// Create log entry for AccelerationRate
CreateLogMessagePara1 ( Timestamp   := AxesGroup.InternalData.SystemTime,
                        MessageType := MessageType.CMD,
                        Severity    := Severity.DEBUG,
                        MessageCode := 0,
                        MessageText := 'Command.AccelerationRate = {1}',
                        Para1       :=  UINT_TO_STRING(_command.AccelerationRate));
                        
// Create log entry for DecelerationRate
CreateLogMessagePara1 ( Timestamp   := AxesGroup.InternalData.SystemTime,
                        MessageType := MessageType.CMD,
                        Severity    := Severity.DEBUG,
                        MessageCode := 0,
                        MessageText := 'Command.DecelerationRate = {1}',
                        Para1       :=  UINT_TO_STRING(_command.DecelerationRate));

// Create log entry for JerkRate
CreateLogMessagePara1 ( Timestamp   := AxesGroup.InternalData.SystemTime,
                        MessageType := MessageType.CMD,
                        Severity    := Severity.DEBUG,
                        MessageCode := 0,
                        MessageText := 'Command.JerkRate = {1}',
                        Para1       :=  UINT_TO_STRING(_command.JerkRate));

// Create log entry for ToolNo
CreateLogMessagePara1 ( Timestamp   := AxesGroup.InternalData.SystemTime,
                        MessageType := MessageType.CMD,
                        Severity    := Severity.DEBUG,
                        MessageCode := 0,
                        MessageText := 'Command.ToolNo = {1}',
                        Para1       :=  USINT_TO_STRING(_command.ToolNo));

// Create log entry for FrameNo
CreateLogMessagePara1 ( Timestamp   := AxesGroup.InternalData.SystemTime,
                        MessageType := MessageType.CMD,
                        Severity    := Severity.DEBUG,
                        MessageCode := 0,
                        MessageText := 'Command.FrameNo = {1}',
                        Para1       :=  USINT_TO_STRING(_command.FrameNo));

// Create log entry for BlendingMode
CreateLogMessagePara1 ( Timestamp   := AxesGroup.InternalData.SystemTime,
                        MessageType := MessageType.CMD,
                        Severity    := Severity.DEBUG,
                        MessageCode := 0,
                        MessageText := 'Command.BlendingMode = {1}',
                        Para1       :=  BLENDING_MODE_TO_STRING(_command.BlendingMode));

// Create log entry for Reserve
CreateLogMessagePara1 ( Timestamp   := AxesGroup.InternalData.SystemTime,
                        MessageType := MessageType.CMD,
                        Severity    := Severity.DEBUG,
                        MessageCode := 0,
                        MessageText := 'Command.Reserve = {1}',
                        Para1       :=  BYTE_TO_STRING(_command.Reserve));

// Create log entry for BlendingParameter[0]
CreateLogMessagePara1 ( Timestamp   := AxesGroup.InternalData.SystemTime,
                        MessageType := MessageType.CMD,
                        Severity    := Severity.DEBUG,
                        MessageCode := 0,
                        MessageText := 'Command.BlendingParameter[0] = {1}',
                        Para1       :=  REAL_TO_STRING(_command.BlendingParameter[0]));

// Create log entry for BlendingParameter[1]
CreateLogMessagePara1 ( Timestamp   := AxesGroup.InternalData.SystemTime,
                        MessageType := MessageType.CMD,
                        Severity    := Severity.DEBUG,
                        MessageCode := 0,
                        MessageText := 'Command.BlendingParameter[1] = {1}',
                        Para1       :=  REAL_TO_STRING(_command.BlendingParameter[1]));

// Create log entry for Position.X
CreateLogMessagePara1 ( Timestamp   := AxesGroup.InternalData.SystemTime,
                        MessageType := MessageType.CMD,
                        Severity    := Severity.DEBUG,
                        MessageCode := 0,
                        MessageText := 'Command.Position.X = {1}',
                        Para1       :=  REAL_TO_STRING(_command.Position.X));

// Create log entry for Position.Y
CreateLogMessagePara1 ( Timestamp   := AxesGroup.InternalData.SystemTime,
                        MessageType := MessageType.CMD,
                        Severity    := Severity.DEBUG,
                        MessageCode := 0,
                        MessageText := 'Command.Position.Y = {1}',
                        Para1       :=  REAL_TO_STRING(_command.Position.Y));

// Create log entry for Position.Z
CreateLogMessagePara1 ( Timestamp   := AxesGroup.InternalData.SystemTime,
                        MessageType := MessageType.CMD,
                        Severity    := Severity.DEBUG,
                        MessageCode := 0,
                        MessageText := 'Command.Position.Z = {1}',
                        Para1       :=  REAL_TO_STRING(_command.Position.Z));

// Create log entry for Position.Rx
CreateLogMessagePara1 ( Timestamp   := AxesGroup.InternalData.SystemTime,
                        MessageType := MessageType.CMD,
                        Severity    := Severity.DEBUG,
                        MessageCode := 0,
                        MessageText := 'Command.Position.Rx = {1}',
                        Para1       :=  REAL_TO_STRING(_command.Position.Rx));

// Create log entry for Position.Ry
CreateLogMessagePara1 ( Timestamp   := AxesGroup.InternalData.SystemTime,
                        MessageType := MessageType.CMD,
                        Severity    := Severity.DEBUG,
                        MessageCode := 0,
                        MessageText := 'Command.Position.Ry = {1}',
                        Para1       :=  REAL_TO_STRING(_command.Position.Ry));

// Create log entry for Position.Rz
CreateLogMessagePara1 ( Timestamp   := AxesGroup.InternalData.SystemTime,
                        MessageType := MessageType.CMD,
                        Severity    := Severity.DEBUG,
                        MessageCode := 0,
                        MessageText := 'Command.Position.Rz = {1}',
                        Para1       :=  REAL_TO_STRING(_command.Position.Rz));

// Create log entry for Position.Config
CreateLogMessagePara1 ( Timestamp   := AxesGroup.InternalData.SystemTime,
                        MessageType := MessageType.CMD,
                        Severity    := Severity.DEBUG,
                        MessageCode := 0,
                        MessageText := 'Command.Config = {1}',
                        Para1       :=  ARM_CONFIG_TO_STRING(_command.Position.Config));

// Create log entry for Position.Reserve
CreateLogMessagePara1 ( Timestamp   := AxesGroup.InternalData.SystemTime,
                        MessageType := MessageType.CMD,
                        Severity    := Severity.DEBUG,
                        MessageCode := 0,
                        MessageText := 'Command.Position.Reserve = {1}',
                        Para1       :=  BYTE_TO_STRING(_command.Reserve));

// Create log entry for Position.TurnNumber[0]
CreateLogMessagePara1 ( Timestamp   := AxesGroup.InternalData.SystemTime,
                        MessageType := MessageType.CMD,
                        Severity    := Severity.DEBUG,
                        MessageCode := 0,
                        MessageText := 'Command.Position.TurnNumber[0] = {1}',
                        Para1       :=  BYTE_TO_STRING(CombineHalfSints(HalfSintHi := _command.Position.TurnNumber.J2Turns, 
                                                                        HalfSintLo := _command.Position.TurnNumber.J1Turns)));

// Create log entry for Position.TurnNumber[1]
CreateLogMessagePara1 ( Timestamp   := AxesGroup.InternalData.SystemTime,
                        MessageType := MessageType.CMD,
                        Severity    := Severity.DEBUG,
                        MessageCode := 0,
                        MessageText := 'Command.Position.TurnNumber[1] = {1}',
                        Para1       :=  BYTE_TO_STRING(CombineHalfSints(HalfSintHi := _command.Position.TurnNumber.J4Turns,
                                                                        HalfSintLo := _command.Position.TurnNumber.J3Turns)));

// Create log entry for Position.TurnNumber[2]
CreateLogMessagePara1 ( Timestamp   := AxesGroup.InternalData.SystemTime,
                        MessageType := MessageType.CMD,
                        Severity    := Severity.DEBUG,
                        MessageCode := 0,
                        MessageText := 'Command.Position.TurnNumber[2] = {1}',
                        Para1       :=  BYTE_TO_STRING(CombineHalfSints(HalfSintHi := _command.Position.TurnNumber.J6Turns,
                                                                        HalfSintLo := _command.Position.TurnNumber.J5Turns)));


// Create log entry for Position.TurnNumber[3]
CreateLogMessagePara1 ( Timestamp   := AxesGroup.InternalData.SystemTime,
                        MessageType := MessageType.CMD,
                        Severity    := Severity.DEBUG,
                        MessageCode := 0,
                        MessageText := 'Command.Position.TurnNumber[3] = {1}',
                        Para1       :=  SINT_TO_STRING(_command.Position.TurnNumber.E1Turns));

// Create log entry for Position.E1
CreateLogMessagePara1 ( Timestamp   := AxesGroup.InternalData.SystemTime,
                        MessageType := MessageType.CMD,
                        Severity    := Severity.DEBUG,
                        MessageCode := 0,
                        MessageText := 'Command.Position.E1 = {1}',
                        Para1       :=  REAL_TO_STRING(_command.Position.E1));

// Create log entry for Manipulation
CreateLogMessagePara1 ( Timestamp   := AxesGroup.InternalData.SystemTime,
                        MessageType := MessageType.CMD,
                        Severity    := Severity.DEBUG,
                        MessageCode := 0,
                        MessageText := 'Command.Manipulation = {1}',
                        Para1       :=  BOOL_TO_STRING(_command.Manipulation));

// Create log entry for TurnMode
CreateLogMessagePara1 ( Timestamp   := AxesGroup.InternalData.SystemTime,
                        MessageType := MessageType.CMD,
                        Severity    := Severity.DEBUG,
                        MessageCode := 0,
                        MessageText := 'Command.TurnMode = {1}',
                        Para1       :=  TURN_MODE_TO_STRING(_command.TurnMode));

// Create log entry for ConfigMode[0]
CreateLogMessagePara1 ( Timestamp   := AxesGroup.InternalData.SystemTime,
                        MessageType := MessageType.CMD,
                        Severity    := Severity.DEBUG,
                        MessageCode := 0,
                        MessageText := 'Command.ConfigMode[0] = {1}',
                        Para1       :=  BYTE_TO_STRING_BIN(_command.ConfigMode[0]));

// Create log entry for ConfigMode[1]
CreateLogMessagePara1 ( Timestamp   := AxesGroup.InternalData.SystemTime,
                        MessageType := MessageType.CMD,
                        Severity    := Severity.DEBUG,
                        MessageCode := 0,
                        MessageText := 'Command.ConfigMode[1] = {1}',
                        Para1       :=  BYTE_TO_STRING_BIN(_command.ConfigMode[1]));

// Create log entry for Reserve3
CreateLogMessagePara1 ( Timestamp   := AxesGroup.InternalData.SystemTime,
                        MessageType := MessageType.CMD,
                        Severity    := Severity.DEBUG,
                        MessageCode := 0,
                        MessageText := 'Command.Reserve3 = {1}',
                        Para1       :=  BYTE_TO_STRING(_command.Reserve3));

// Create log entry for Reserve4
CreateLogMessagePara1 ( Timestamp   := AxesGroup.InternalData.SystemTime,
                        MessageType := MessageType.CMD,
                        Severity    := Severity.DEBUG,
                        MessageCode := 0,
                        MessageText := 'Command.Reserve4 = {1}',
                        Para1       :=  BYTE_TO_STRING(_command.Reserve4));

// Create log entry for MoveTime
CreateLogMessagePara1 ( Timestamp   := AxesGroup.InternalData.SystemTime,
                        MessageType := MessageType.CMD,
                        Severity    := Severity.DEBUG,
                        MessageCode := 0,
                        MessageText := 'Command.MoveTime = {1}',
                        Para1       :=  UINT_TO_STRING(_command.MoveTime));

// Create log entry for Position.E2
CreateLogMessagePara1 ( Timestamp   := AxesGroup.InternalData.SystemTime,
                        MessageType := MessageType.CMD,
                        Severity    := Severity.DEBUG,
                        MessageCode := 0,
                        MessageText := 'Command.Position.E2 = {1}',
                        Para1       :=  REAL_TO_STRING(_command.Position.E2));

// Create log entry for Position.E3
CreateLogMessagePara1 ( Timestamp   := AxesGroup.InternalData.SystemTime,
                        MessageType := MessageType.CMD,
                        Severity    := Severity.DEBUG,
                        MessageCode := 0,
                        MessageText := 'Command.Position.E3 = {1}',
                        Para1       :=  REAL_TO_STRING(_command.Position.E3));

// Create log entry for Position.E4
CreateLogMessagePara1 ( Timestamp   := AxesGroup.InternalData.SystemTime,
                        MessageType := MessageType.CMD,
                        Severity    := Severity.DEBUG,
                        MessageCode := 0,
                        MessageText := 'Command.Position.E4 = {1}',
                        Para1       :=  REAL_TO_STRING(_command.Position.E4));

// Create log entry for Position.E5
CreateLogMessagePara1 ( Timestamp   := AxesGroup.InternalData.SystemTime,
                        MessageType := MessageType.CMD,
                        Severity    := Severity.DEBUG,
                        MessageCode := 0,
                        MessageText := 'Command.Position.E5 = {1}',
                        Para1       :=  REAL_TO_STRING(_command.Position.E5));

// Create log entry for Position.E6
CreateLogMessagePara1 ( Timestamp   := AxesGroup.InternalData.SystemTime,
                        MessageType := MessageType.CMD,
                        Severity    := Severity.DEBUG,
                        MessageCode := 0,
                        MessageText := 'Command.Position.E6 = {1}',
                        Para1       :=  REAL_TO_STRING(_command.Position.E6));
END_METHOD

METHOD FB_init : BOOL
VAR_INPUT
  /// if TRUE, the retain variables are initialized (warm start / cold start)
  bInitRetains : BOOL; 
  /// if TRUE, the instance afterwards gets moved into the copy code (online change)
  bInCopyCode  : BOOL;  
END_VAR
MyType := 'MC_MoveDirectAbsoluteFB';
END_METHOD

METHOD PROTECTED OnCall
VAR_IN_OUT
  /// Robot assignment of function
  AxesGroup : AxesGroup; 
END_VAR
// call base implementation
SUPER^.OnCall(AxesGroup := AxesGroup);

CASE _stepCmd OF
  
  00:  IF ( _execute_R.Q )  
       THEN
         // Check function is supported and parameter are valid ?
         IF (( CheckFunctionSupported( AxesGroup := AxesGroup )) AND
             ( CheckParameterValid   ( AxesGroup := AxesGroup )))      
         THEN
           // set busy flag
           Busy := TRUE;
           // Reset command outputs
           SysDepMemSet(pDest := ADR(OutCmd), Value := 0, DataLen := SIZEOF(OutCmd));         
           // apply command parameter
          _parCmd := ParCmd;
           // init parameter sequence
          _command.ParSeq := 1;
           // create command data
           CommandData := CreateCommandPayload(AxesGroup := AxesGroup);
           // Add command to active command register
          _uniqueID := AxesGroup.Acyclic.ActiveCommandRegister.AddCmd( pCommandFB := ADR(THIS^ ));     
           // set timeout
           SetTimeout(PT := _timeoutCmd, rTimer := _timerCmd);
           // inc step counter
          _stepCmd := _stepCmd + 1;
         END_IF 
       END_IF
     

  01:  // Wait for responce received
       IF ( _responseReceived )
       THEN
         // reset response received flag
        _responseReceived := FALSE;
         // reset Active flag
         Active := FALSE;
         
         CASE  _response.State 
         OF
           CmdMessageState.BUFFERED    : CommandBuffered    := TRUE;
           CmdMessageState.ACTIVE      : Active             := TRUE;
           CmdMessageState.INTERRUPTED : CommandInterrupted := TRUE;           
           CmdMessageState.DONE        : Done               := TRUE;           
           CmdMessageState.ABORTED     : CommandAborted     := TRUE;
           CmdMessageState.ERROR       : Error              := TRUE;
         END_CASE
                
         // Done, Aborted or Error ?
         IF (_response.State >= CmdMessageState.DONE )
         THEN
           // Reset Busy flag
           Busy := FALSE;
           // Update results
           OutCmd.Progress          := _response.Progress;
           OutCmd.FollowID          := _response.OriginID;
           OutCmd.RemainingDistance := _response.RemainingDistance;
           // set timeout
           SetTimeout(PT := _timeoutCmd, rTimer := _timerCmd);
           // inc step counter
          _stepCmd := _stepCmd + 1; 
         END_IF
       END_IF


  02: IF ( NOT Execute)
      THEN
        Reset();
      END_IF     

ELSE
  // invalid step
  ErrorID := RobotLibraryEvents.ERR_INVALID_STEP;
END_CASE


// Reset FB
IF ( NOT Execute )
THEN
  Reset();
END_IF
END_METHOD

METHOD INTERNAL ParseResponsePayload : DINT
VAR_INPUT
  /// Response data
  ResponseData : RobotLibraryRecvDataFB;
  /// Timestamp
  Timestamp    : SystemTime;  
END_VAR
// Table 6-255: Received CMD payload (RC to PLC) of "MoveDirectAbsolute"
// --------------------------
// Header
// --------------------------
// Byte 00 : USINT   - ParSeq | State     
// Byte 01 : SINT    - AlarmMessageSeverity    
// Byte 02 : UINT    - AlarmMessageCode HB
// Byte 03 :         - AlarmMessageCode LB
// --------------------------
// Datablock
// --------------------------
// Byte 04 : USINT      - InvocationCounter
// Byte 05 : SINT       - Reserved
// Byte 06 : INT        - OriginID HW HB
// Byte 07 :            - OriginID HW LB
// Byte 08 : UINT       - Progress HW HB
// Byte 09 :            - Progress HW LB
// Byte 10 : REAL       - RemainingDistance HW HB
// Byte 11 :            - RemainingDistance HW LB
// Byte 12 :            - RemainingDistance LW HB
// Byte 13 :            - RemainingDistance LW LB
// call base implementation to parse the header from payload buffer
ResponseData.PayloadPtr := SUPER^.ParseResponsePayload(ResponseData := ResponseData, Timestamp := Timestamp);

// copy parsed header to response
_response.ParSeq               := _rspHeader.ParSeq;
_response.State                := _rspHeader.State;
_response.AlarmMessageSeverity := _rspHeader.AlarmMessageSeverity;
_response.AlarmMessageCode     := _rspHeader.AlarmMessageCode;

// Get Response.InvocationCounter
_response.InvocationCounter := ResponseData.GetUsint();
// Get Response.Reserve
_response.Reserve := ResponseData.GetSint();
// Get Response.OriginID
_response.OriginID := ResponseData.GetInt();
// Get Response.Progress
_response.Progress := ResponseData.GetUint();
// Get Response.RemainingDistance
_response.RemainingDistance := ResponseData.GetReal();

// Create logging
ParseResponsePayloadLog(ResponseData := ResponseData, Timestamp := Timestamp);
END_METHOD

METHOD INTERNAL ParseResponsePayloadLog
VAR_INPUT
  /// Response data
  ResponseData : RobotLibraryRecvDataFB;
  /// Timestamp
  Timestamp    : SystemTime;  
END_VAR
// Create log entry for Parameter start
CreateLogMessage      ( Timestamp   := Timestamp,
                        MessageType := MessageType.CMD,
                        Severity    := Severity.DEBUG,
                        MessageCode := 0,
                        MessageText := 'Parsed the following parameter(s) from response data:');
                        
// Create log entry for InvocationCounter
CreateLogMessagePara1 ( Timestamp   := Timestamp,
                        MessageType := MessageType.CMD,
                        Severity    := Severity.DEBUG,
                        MessageCode := 0,
                        MessageText := 'Response.InvocationCounter = {1}',
                        Para1       :=  USINT_TO_STRING(_response.InvocationCounter));

// Create log entry for Reserve
CreateLogMessagePara1 ( Timestamp   := Timestamp,
                        MessageType := MessageType.CMD,
                        Severity    := Severity.DEBUG,
                        MessageCode := 0,
                        MessageText := 'Response.Reserve = {1}',
                        Para1       :=  SINT_TO_STRING(_response.Reserve));

// Create log entry for OriginID
CreateLogMessagePara1 ( Timestamp   := Timestamp,
                        MessageType := MessageType.CMD,
                        Severity    := Severity.DEBUG,
                        MessageCode := 0,
                        MessageText := 'Response.OriginID = {1}',
                        Para1       :=  INT_TO_STRING(_response.OriginID));

// Create log entry for Progress
CreateLogMessagePara1 ( Timestamp   := Timestamp,
                        MessageType := MessageType.CMD,
                        Severity    := Severity.DEBUG,
                        MessageCode := 0,
                        MessageText := 'Response.Progress = {1}',
                        Para1       :=  UINT_TO_STRING(_response.Progress));

// Create log entry for RemainingDistance
CreateLogMessagePara1 ( Timestamp   := Timestamp,
                        MessageType := MessageType.CMD,
                        Severity    := Severity.DEBUG,
                        MessageCode := 0,
                        MessageText := 'Response.RemainingDistance = {1}',
                        Para1       :=  REAL_TO_STRING(_response.RemainingDistance));
END_METHOD

METHOD PROTECTED Reset : DINT
VAR_INPUT
END_VAR
Reset := SUPER^.Reset();

Done               := FALSE;
Busy               := FALSE;
Active             := FALSE;
CommandBuffered    := FALSE;
CommandAborted     := FALSE;
CommandInterrupted := FALSE;
END_METHOD

END_FUNCTION_BLOCK

// Library/POUs/BasicMove/MC_MoveLinearAbsolute/MC_MoveLinearAbsoluteFB
/// Move the TCP to an absolute cartesian position (linear interpolation)
FUNCTION_BLOCK MC_MoveLinearAbsoluteFB EXTENDS RobotLibraryBaseExecuteFB
// ------------------------------------------------------------------------- 
//  SRCI Robot Library                                                
// ------------------------------------------------------------------------- 
//                                                                           
//  Object:      MoveLinearAbsoluteFB                                       
//  Author:      Thorsten Brach                                                
//  Date:        2024-06-01
//
//  Description:                                              
//   
//                                                                           
//  Copyright: 
//    (C) 2024 Thorsten Brach. All rights reserved                                                                                                                                            
//             Licensed under the LGPL-3.0 license.
//                                                                           
//  Disclaimer:                                                                           
//    This project is provided without any guarantee and can be used for   
//    private and commercial purposes. Any use is at the user’s 
//    own risk and responsibility.
//
// -------------------------------------------------------------------------
VAR_INPUT
  /// Parameter which determines the behavior towards the previously sent and still active or buffered commands
  AbortingMode       : AbortingMode;
  /// Defines the target sequence in which the command will be executed
  SequenceFlag       : SequenceFlag;
  /// command outputs
  ParCmd             : MoveLinearAbsoluteParCmd;       
END_VAR

VAR_OUTPUT
  /// Command is transferred and confirmed by the RC
  CommandBuffered    : BOOL;
  /// The command takes control of the motion of the according axis group
  Active             : BOOL;
  /// The command was aborted by another command.
  CommandAborted     : BOOL;
  /// TRUE, while command is interrupted during execution and can be continued
  CommandInterrupted : BOOL;
  /// command outputs
  OutCmd             : MoveLinearAbsoluteOutCmd;       
END_VAR



VAR
  /// internal copy of command parameter 
 _parCmd             : MoveLinearAbsoluteParCmd;
  /// command data to send
 _command            : MoveLinearAbsoluteSendData;
  /// response data received
 _response           : MoveLinearAbsoluteRecvData;      
END_VAR

SUPER^(AxesGroup := AxesGroup);

METHOD PROTECTED CheckFunctionSupported : BOOL
VAR_IN_OUT
  /// Robot assignment of function
  AxesGroup : AxesGroup; 
END_VAR
CheckFunctionSupported := AxesGroup.InternalData.RCSupportedFunctions.MoveLinearAbsolute;

IF ( NOT CheckFunctionSupported )
THEN
  // call base implementation for set error and create log entry
  SUPER^.CheckFunctionSupported(AxesGroup := AxesGroup);
END_IF
END_METHOD

METHOD PROTECTED CheckParameterChanged : BOOL
VAR_IN_OUT
  /// Robot assignment of function
  AxesGroup    : AxesGroup; 
END_VAR
// Check ParCmd Size is > 0, because MemCmp does not work correctly with size = 0
IF (SIZEOF(ParCmd) = 0) 
THEN 
  RETURN;
END_IF

// compare memory 
_parameterChanged := ( SysDepMemCmp(pData1 := ADR(ParCmd), pData2 := ADR(_parCmd), DataLen := SIZEOF(ParCmd)) <> RobotLibraryConstants.OK );

// check parameter valid ?
_parameterValid   := CheckParameterValid( AxesGroup := AxesGroup );

IF ((  _parameterChanged        )  AND 
    (  _parameterValid          )) OR
    (  _parameterUpdateInternal )  
THEN  
  // reset internal flag for send parameter update
 _parameterUpdateInternal := FALSE;
  // update internal copy of parameters 
 _parCmd := ParCmd;
  // inc parameter sequence
 _command.ParSeq := _command.ParSeq + 1;
  // update command data  
  CommandData := CreateCommandPayload(AxesGroup := AxesGroup); // ( Access via reference to rCommandFB in ACR )
  // notify active command register 
  AxesGroup.Acyclic.ActiveCommandRegister.NotifyParameterChanged := _uniqueID;
END_IF
END_METHOD

METHOD INTERNAL CreateCommandPayload : RobotLibrarySendDataFB
VAR_IN_OUT
  /// Robot assignment of function
  AxesGroup : AxesGroup; 
END_VAR
// Table 6-245: Sent CMD payload (PLC to RC) of "MoveLinearAbsolute"
// --------------------------
// Header
// --------------------------
// Byte 00 : UINT  - Type HB     
// Byte 01 :       - Type LB    
// Byte 02 : USINT - Reserve | ExecutionMode
// Byte 03 : USINT - ParSeq  | Priority
// --------------------------
// Datablock
// --------------------------
// Byte 04 : SINT       - EmitterID[0]
// Byte 05 : SINT       - EmitterID[1]
// Byte 06 : SINT       - EmitterID[2]
// Byte 07 : SINT       - EmitterID[3]
// Byte 08 : SINT       - ListenerID
// Byte 09 : BYTE       - Reserved
// Byte 10 : UINT       - VelocityRate HW HB
// Byte 11 :            - VelocityRate HW LB
// Byte 12 : UINT       - AccelerationRate HW HB
// Byte 13 :            - AccelerationRate HW LB
// Byte 14 : UINT       - DecelerationRate HW HB
// Byte 15 :            - DecelerationRate HW LB
// Byte 16 : UINT       - JerkRate HW HB
// Byte 17 :            - JerkRate HW LB
// Byte 18 : USINT      - ToolNo
// Byte 19 : USINT      - FrameNo
// Byte 20 : USINT      - BlendingMode
// Byte 21 : USINT      - OriMode
// Byte 22 : REAL       - BlendingParameter[0] HW HB
// Byte 23 :            - BlendingParameter[0] HW LB
// Byte 24 :            - BlendingParameter[0] LW HB
// Byte 25 :            - BlendingParameter[0] LW LB
// Byte 26 : REAL       - BlendingParameter[1] HW HB
// Byte 27 :            - BlendingParameter[1] HW LB
// Byte 28 :            - BlendingParameter[1] LW HB
// Byte 29 :            - BlendingParameter[1] LW LB
// Byte 30 : REAL       - Position.X HW HB
// Byte 31 :            - Position.X HW LB
// Byte 32 :            - Position.X LW HB
// Byte 33 :            - Position.X LW LB
// Byte 34 : REAL       - Position.Y HW HB
// Byte 35 :            - Position.Y HW LB
// Byte 36 :            - Position.Y LW HB
// Byte 37 :            - Position.Y LW LB
// Byte 38 : REAL       - Position.Z HW HB
// Byte 39 :            - Position.Z HW LB
// Byte 40 :            - Position.Z LW HB
// Byte 41 :            - Position.Z LW LB
// Byte 42 : REAL       - Position.RX HW HB
// Byte 43 :            - Position.RX HW LB
// Byte 44 :            - Position.RX LW HB
// Byte 45 :            - Position.RX LW LB
// Byte 46 : REAL       - Position.RY HW HB
// Byte 47 :            - Position.RY HW LB
// Byte 48 :            - Position.RY LW HB
// Byte 49 :            - Position.RY LW LB
// Byte 50 : REAL       - Position.RZ HW HB
// Byte 51 :            - Position.RZ HW LB
// Byte 52 :            - Position.RZ LW HB
// Byte 53 :            - Position.RZ LW LB
// Byte 54 : BYTE       - - - - - W E S
// Byte 55 : BYTE       - Reserved
// Byte 56 : BYTE       - Position.TurnNumber[0]
// Byte 57 : BYTE       - Position.TurnNumber[1]
// Byte 58 : BYTE       - Position.TurnNumber[2]
// Byte 59 : BYTE       - Position.TurnNumber[3]
// Byte 60 : REAL       - Position.E1 HW HB
// Byte 61 :            - Position.E1 HW LB
// Byte 62 :            - Position.E1 LW HB
// Byte 63 :            - Position.E1 LW LB
// Byte 64 : BOOL       - Manipulation
// Byte 65 : USINT      - TurnMode
// Byte 66 : BYTE       - ConfigMode[0]
// Byte 67 : BYTE       - ConfigMode[1]
// Byte 68 : BYTE       - Reserved
// Byte 69 : BYTE       - Reserved
// Byte 70 : UINT       - Time HW HB
// Byte 71 :            - Time HW LB
// Byte 72 : REAL       - Position.E2 HW HB
// Byte 73 :            - Position.E2 HW LB
// Byte 74 :            - Position.E2 LW HB
// Byte 75 :            - Position.E2 LW LB
// Byte 76 : REAL       - Position.E3 HW HB
// Byte 77 :            - Position.E3 HW LB
// Byte 78 :            - Position.E3 LW HB
// Byte 79 :            - Position.E3 LW LB
// Byte 80 : REAL       - Position.E4 HW HB
// Byte 81 :            - Position.E4 HW LB
// Byte 82 :            - Position.E4 LW HB
// Byte 83 :            - Position.E4 LW LB
// Byte 84 : REAL       - Position.E5 HW HB
// Byte 85 :            - Position.E5 HW LB
// Byte 86 :            - Position.E5 LW HB
// Byte 87 :            - Position.E5 LW LB
// Byte 88 : REAL       - Position.E6 HW HB
// Byte 89 :            - Position.E6 HW LB
// Byte 90 :            - Position.E6 LW HB
// Byte 91 :            - Position.E6 LW LB
// --------------------------
// set command parameter 
_command.CmdTyp            :=  CmdType.MoveLinearAbsolute;
_command.ExecMode          :=  ExecMode;
_command.ParSeq            := _command.ParSeq;
_command.Priority          :=  Priority;
_command.EmitterID         := _parCmd.EmitterID;
_command.Reserve           :=  0;
_command.ListenerID        :=  0; {warning 'ToDo'}
_command.Reserve           :=  0;
_command.VelocityRate      :=  REAL_TO_PERCENT_UINT(_parCmd.VelocityRate     , IsOptional := FALSE);
_command.AccelerationRate  :=  REAL_TO_PERCENT_UINT(_parCmd.AccelerationRate , IsOptional := FALSE);
_command.JerkRate          :=  REAL_TO_PERCENT_UINT(_parCmd.JerkRate         , IsOptional := TRUE );
_command.DecelerationRate  :=  REAL_TO_PERCENT_UINT(_parCmd.DecelerationRate , IsOptional := TRUE );
_command.ToolNo            := _parCmd.ToolNo;
_command.FrameNo           := _parCmd.FrameNo;
_command.BlendingMode      := _parCmd.BlendingMode;
_command.OriMode           := _parcmd.OriMode;
_command.BlendingParameter := _parCmd.BlendingParameter;
_command.Position          := _parCmd.Position;
_command.Manipulation      := _parCmd.Manipulation;
_command.TurnMode          := _parCmd.TurnMode;
_command.ConfigMode        :=  ArmConfigParameterToBytes(_parCmd.ConfigMode);
_command.Reserve2          := 0;
_command.Reserve3          := 0;
_command.MoveTime          := TIME_TO_UINT(_parCmd.MoveTime);


// copy command data to header
_cmdHeader := _command;
// call base implementation to copy header to payload buffer
CreateCommandPayload := SUPER^.CreateCommandPayload(AxesGroup := AxesGroup);

// add command.EmitterID[0]
CreateCommandPayload.AddSint(_command.EmitterID[0]);
// add command.EmitterID[1]
CreateCommandPayload.AddSint(_command.EmitterID[1]);
// add command.EmitterID[2]
CreateCommandPayload.AddSint(_command.EmitterID[2]);
// add command.EmitterID[3]
CreateCommandPayload.AddSint(_command.EmitterID[3]);
// add command.ListenerID
CreateCommandPayload.AddSint(_command.ListenerID);
// add command.Reserve
CreateCommandPayload.AddByte(_command.Reserve);
// add command.VelocityRate
CreateCommandPayload.AddUint(_command.VelocityRate);
// add command.AccelerationRate
CreateCommandPayload.AddUint(_command.AccelerationRate);
// add command.DecelerationRate
CreateCommandPayload.AddUint(_command.DecelerationRate);
// add command.JerkRate
CreateCommandPayload.AddUint(_command.JerkRate);
// add command.ToolNo
CreateCommandPayload.AddUsint(_command.ToolNo);
// add command.mFrameNo
CreateCommandPayload.AddUsint(_command.FrameNo);
// add command.BlendingMode
CreateCommandPayload.AddUsint(_command.BlendingMode);
// add command.OriMode
CreateCommandPayload.AddUsint(_command.OriMode);
// add command.BlendingParameter[0]
CreateCommandPayload.AddReal(_command.BlendingParameter[0]);
// add command.BlendingParameter[1]
CreateCommandPayload.AddReal(_command.BlendingParameter[1]);
// add command.Position.X
CreateCommandPayload.AddReal(_command.Position.X);
// add command.Position.Y
CreateCommandPayload.AddReal(_command.Position.Y);
// add command.Position.Z
CreateCommandPayload.AddReal(_command.Position.Z);
// add command.Position.Rx
CreateCommandPayload.AddReal(_command.Position.Rx);
// add command.Position.Ry
CreateCommandPayload.AddReal(_command.Position.Ry);
// add command.Position.Rz
CreateCommandPayload.AddReal(_command.Position.Rz);
// add command.Position.Config
CreateCommandPayload.AddArmConfig(_command.Position.Config);
// add command.Position.TurnNumber
CreateCommandPayload.AddTurnNumber(_command.Position.TurnNumber);
// add command.Position.E1
CreateCommandPayload.AddReal(_command.Position.E1);
// add command.Manipulation
CreateCommandPayload.AddBool(_command.Manipulation);
// add command.TurnMode
CreateCommandPayload.AddUsint(_command.TurnMode);
// add command.ConfigMode[0]
CreateCommandPayload.AddByte(_command.ConfigMode[0]);
// add command.ConfigMode[1]
CreateCommandPayload.AddByte(_command.ConfigMode[1]);
// add command.Reserve2
CreateCommandPayload.AddByte(_command.Reserve2);
// add command.Reserve3
CreateCommandPayload.AddByte(_command.Reserve3);
// add command.MoveTime
CreateCommandPayload.AddUint(_command.MoveTime);
// add command.Position.E2
CreateCommandPayload.AddReal(_command.Position.E2);
// add command.Position.E3
CreateCommandPayload.AddReal(_command.Position.E3);
// add command.Position.E4
CreateCommandPayload.AddReal(_command.Position.E4);
// add command.Position.E5
CreateCommandPayload.AddReal(_command.Position.E5);
// add command.Position.E6
CreateCommandPayload.AddReal(_command.Position.E6);

// Create logging
CreateCommandPayloadLog(AxesGroup := AxesGroup);
END_METHOD

METHOD INTERNAL CreateCommandPayloadLog 
VAR_IN_OUT
  /// Robot assignment of function
  AxesGroup : AxesGroup; 
END_VAR
VAR 
  /// internal index for loops
 _idx : DINT;
END_VAR
// Create log entry for Parameter start
CreateLogMessage      ( Timestamp   := AxesGroup.InternalData.SystemTime,
                        MessageType := MessageType.CMD,
                        Severity    := Severity.DEBUG,
                        MessageCode := 0,
                        MessageText := 'Create command payload with the following parameter(s) :');

// Create log entry for EmitterID[x]
FOR _idx := 0 TO 3
DO
  CreateLogMessagePara2 ( Timestamp   := AxesGroup.InternalData.SystemTime,
                          MessageType := MessageType.CMD,
                          Severity    := Severity.DEBUG,
                          MessageCode := 0,
                          MessageText := 'Command.EmitterID[{2}] = {1}',
                          Para1       :=  SINT_TO_STRING(_command.EmitterID[_idx]),
                          Para2       :=  DINT_TO_STRING(_idx));
END_FOR

// Create log entry for ListenerID
CreateLogMessagePara1 ( Timestamp   := AxesGroup.InternalData.SystemTime,
                        MessageType := MessageType.CMD,
                        Severity    := Severity.DEBUG,
                        MessageCode := 0,
                        MessageText := 'Command.ListenerID = {1}',
                        Para1       :=  SINT_TO_STRING(_command.ListenerID));

// Create log entry for Reserve
CreateLogMessagePara1 ( Timestamp   := AxesGroup.InternalData.SystemTime,
                        MessageType := MessageType.CMD,
                        Severity    := Severity.DEBUG,
                        MessageCode := 0,
                        MessageText := 'Command.Reserve = {1}',
                        Para1       :=  BYTE_TO_STRING(_command.Reserve));


// Create log entry for VelocityRate
CreateLogMessagePara1 ( Timestamp   := AxesGroup.InternalData.SystemTime,
                        MessageType := MessageType.CMD,
                        Severity    := Severity.DEBUG,
                        MessageCode := 0,
                        MessageText := 'Command.VelocityRate = {1}',
                        Para1       :=  UINT_TO_STRING(_command.VelocityRate));

// Create log entry for AccelerationRate
CreateLogMessagePara1 ( Timestamp   := AxesGroup.InternalData.SystemTime,
                        MessageType := MessageType.CMD,
                        Severity    := Severity.DEBUG,
                        MessageCode := 0,
                        MessageText := 'Command.AccelerationRate = {1}',
                        Para1       :=  UINT_TO_STRING(_command.AccelerationRate));
                        
// Create log entry for DecelerationRate
CreateLogMessagePara1 ( Timestamp   := AxesGroup.InternalData.SystemTime,
                        MessageType := MessageType.CMD,
                        Severity    := Severity.DEBUG,
                        MessageCode := 0,
                        MessageText := 'Command.DecelerationRate = {1}',
                        Para1       :=  UINT_TO_STRING(_command.DecelerationRate));

// Create log entry for JerkRate
CreateLogMessagePara1 ( Timestamp   := AxesGroup.InternalData.SystemTime,
                        MessageType := MessageType.CMD,
                        Severity    := Severity.DEBUG,
                        MessageCode := 0,
                        MessageText := 'Command.JerkRate = {1}',
                        Para1       :=  UINT_TO_STRING(_command.JerkRate));

// Create log entry for ToolNo
CreateLogMessagePara1 ( Timestamp   := AxesGroup.InternalData.SystemTime,
                        MessageType := MessageType.CMD,
                        Severity    := Severity.DEBUG,
                        MessageCode := 0,
                        MessageText := 'Command.ToolNo = {1}',
                        Para1       :=  USINT_TO_STRING(_command.ToolNo));

// Create log entry for FrameNo
CreateLogMessagePara1 ( Timestamp   := AxesGroup.InternalData.SystemTime,
                        MessageType := MessageType.CMD,
                        Severity    := Severity.DEBUG,
                        MessageCode := 0,
                        MessageText := 'Command.FrameNo = {1}',
                        Para1       :=  USINT_TO_STRING(_command.FrameNo));

// Create log entry for BlendingMode
CreateLogMessagePara1 ( Timestamp   := AxesGroup.InternalData.SystemTime,
                        MessageType := MessageType.CMD,
                        Severity    := Severity.DEBUG,
                        MessageCode := 0,
                        MessageText := 'Command.BlendingMode = {1}',
                        Para1       :=  BLENDING_MODE_TO_STRING(_command.BlendingMode));

// Create log entry for OriMode
CreateLogMessagePara1 ( Timestamp   := AxesGroup.InternalData.SystemTime,
                        MessageType := MessageType.CMD,
                        Severity    := Severity.DEBUG,
                        MessageCode := 0,
                        MessageText := 'Command.OriMode = {1}',
                        Para1       :=  ORI_MODE_TO_STRING(_command.OriMode));

// Create log entry for BlendingParameter[0]
CreateLogMessagePara1 ( Timestamp   := AxesGroup.InternalData.SystemTime,
                        MessageType := MessageType.CMD,
                        Severity    := Severity.DEBUG,
                        MessageCode := 0,
                        MessageText := 'Command.BlendingParameter[0] = {1}',
                        Para1       :=  REAL_TO_STRING(_command.BlendingParameter[0]));

// Create log entry for BlendingParameter[1]
CreateLogMessagePara1 ( Timestamp   := AxesGroup.InternalData.SystemTime,
                        MessageType := MessageType.CMD,
                        Severity    := Severity.DEBUG,
                        MessageCode := 0,
                        MessageText := 'Command.BlendingParameter[1] = {1}',
                        Para1       :=  REAL_TO_STRING(_command.BlendingParameter[1]));

// Create log entry for Position.X
CreateLogMessagePara1 ( Timestamp   := AxesGroup.InternalData.SystemTime,
                        MessageType := MessageType.CMD,
                        Severity    := Severity.DEBUG,
                        MessageCode := 0,
                        MessageText := 'Command.Position.X = {1}',
                        Para1       :=  REAL_TO_STRING(_command.Position.X));

// Create log entry for Position.Y
CreateLogMessagePara1 ( Timestamp   := AxesGroup.InternalData.SystemTime,
                        MessageType := MessageType.CMD,
                        Severity    := Severity.DEBUG,
                        MessageCode := 0,
                        MessageText := 'Command.Position.Y = {1}',
                        Para1       :=  REAL_TO_STRING(_command.Position.Y));

// Create log entry for Position.Z
CreateLogMessagePara1 ( Timestamp   := AxesGroup.InternalData.SystemTime,
                        MessageType := MessageType.CMD,
                        Severity    := Severity.DEBUG,
                        MessageCode := 0,
                        MessageText := 'Command.Position.Z = {1}',
                        Para1       :=  REAL_TO_STRING(_command.Position.Z));

// Create log entry for Position.Rx
CreateLogMessagePara1 ( Timestamp   := AxesGroup.InternalData.SystemTime,
                        MessageType := MessageType.CMD,
                        Severity    := Severity.DEBUG,
                        MessageCode := 0,
                        MessageText := 'Command.Position.Rx = {1}',
                        Para1       :=  REAL_TO_STRING(_command.Position.Rx));

// Create log entry for Position.Ry
CreateLogMessagePara1 ( Timestamp   := AxesGroup.InternalData.SystemTime,
                        MessageType := MessageType.CMD,
                        Severity    := Severity.DEBUG,
                        MessageCode := 0,
                        MessageText := 'Command.Position.Ry = {1}',
                        Para1       :=  REAL_TO_STRING(_command.Position.Ry));

// Create log entry for Position.Rz
CreateLogMessagePara1 ( Timestamp   := AxesGroup.InternalData.SystemTime,
                        MessageType := MessageType.CMD,
                        Severity    := Severity.DEBUG,
                        MessageCode := 0,
                        MessageText := 'Command.Position.Rz = {1}',
                        Para1       :=  REAL_TO_STRING(_command.Position.Rz));

// Create log entry for Position.Config
CreateLogMessagePara1 ( Timestamp   := AxesGroup.InternalData.SystemTime,
                        MessageType := MessageType.CMD,
                        Severity    := Severity.DEBUG,
                        MessageCode := 0,
                        MessageText := 'Command.Position.Config = {1}',
                        Para1       :=  ARM_CONFIG_TO_STRING(_command.Position.Config));

// Create log entry for Position.TurnNumber[0]
CreateLogMessagePara1 ( Timestamp   := AxesGroup.InternalData.SystemTime,
                        MessageType := MessageType.CMD,
                        Severity    := Severity.DEBUG,
                        MessageCode := 0,
                        MessageText := 'Command.Position.TurnNumber[0] = {1}',
                        Para1       :=  BYTE_TO_STRING(CombineHalfSints(HalfSintHi := _command.Position.TurnNumber.J2Turns, 
                                                                        HalfSintLo := _command.Position.TurnNumber.J1Turns)));

// Create log entry for Position.TurnNumber[1]
CreateLogMessagePara1 ( Timestamp   := AxesGroup.InternalData.SystemTime,
                        MessageType := MessageType.CMD,
                        Severity    := Severity.DEBUG,
                        MessageCode := 0,
                        MessageText := 'Command.Position.TurnNumber[1] = {1}',
                        Para1       :=  BYTE_TO_STRING(CombineHalfSints(HalfSintHi := _command.Position.TurnNumber.J4Turns, 
                                                                        HalfSintLo := _command.Position.TurnNumber.J3Turns)));

// Create log entry for Position.TurnNumber[2]
CreateLogMessagePara1 ( Timestamp   := AxesGroup.InternalData.SystemTime,
                        MessageType := MessageType.CMD,
                        Severity    := Severity.DEBUG,
                        MessageCode := 0,
                        MessageText := 'Command.Position.TurnNumber[2] = {1}',
                        Para1       :=  BYTE_TO_STRING(CombineHalfSints(HalfSintHi := _command.Position.TurnNumber.J6Turns, 
                                                                        HalfSintLo := _command.Position.TurnNumber.J5Turns)));


// Create log entry for Position.TurnNumber[3]
CreateLogMessagePara1 ( Timestamp   := AxesGroup.InternalData.SystemTime,
                        MessageType := MessageType.CMD,
                        Severity    := Severity.DEBUG,
                        MessageCode := 0,
                        MessageText := 'Command.Position.TurnNumber[3] = {1}',
                        Para1       :=  SINT_TO_STRING(_command.Position.TurnNumber.E1Turns));

// Create log entry for Position.E1
CreateLogMessagePara1 ( Timestamp   := AxesGroup.InternalData.SystemTime,
                        MessageType := MessageType.CMD,
                        Severity    := Severity.DEBUG,
                        MessageCode := 0,
                        MessageText := 'Command.Position.E1 = {1}',
                        Para1       :=  REAL_TO_STRING(_command.Position.E1));

// Create log entry for Manipulation
CreateLogMessagePara1 ( Timestamp   := AxesGroup.InternalData.SystemTime,
                        MessageType := MessageType.CMD,
                        Severity    := Severity.DEBUG,
                        MessageCode := 0,
                        MessageText := 'Command.Manipulation = {1}',
                        Para1       :=  BOOL_TO_STRING(_command.Manipulation));

// Create log entry for TurnMode
CreateLogMessagePara1 ( Timestamp   := AxesGroup.InternalData.SystemTime,
                        MessageType := MessageType.CMD,
                        Severity    := Severity.DEBUG,
                        MessageCode := 0,
                        MessageText := 'Command.TurnMode = {1}',
                        Para1       :=  TURN_MODE_TO_STRING(_command.TurnMode));

// Create log entry for ConfigMode[0]
CreateLogMessagePara1 ( Timestamp   := AxesGroup.InternalData.SystemTime,
                        MessageType := MessageType.CMD,
                        Severity    := Severity.DEBUG,
                        MessageCode := 0,
                        MessageText := 'Command.ConfigMode[0] = {1}',
                        Para1       :=  BYTE_TO_STRING_BIN(_command.ConfigMode[0]));

// Create log entry for ConfigMode[1]
CreateLogMessagePara1 ( Timestamp   := AxesGroup.InternalData.SystemTime,
                        MessageType := MessageType.CMD,
                        Severity    := Severity.DEBUG,
                        MessageCode := 0,
                        MessageText := 'Command.ConfigMode[1] = {1}',
                        Para1       :=  BYTE_TO_STRING_BIN(_command.ConfigMode[1]));

// Create log entry for Reserve2
CreateLogMessagePara1 ( Timestamp   := AxesGroup.InternalData.SystemTime,
                        MessageType := MessageType.CMD,
                        Severity    := Severity.DEBUG,
                        MessageCode := 0,
                        MessageText := 'Command.Reserve2 = {1}',
                        Para1       :=  BYTE_TO_STRING(_command.Reserve2));

// Create log entry for Reserve3
CreateLogMessagePara1 ( Timestamp   := AxesGroup.InternalData.SystemTime,
                        MessageType := MessageType.CMD,
                        Severity    := Severity.DEBUG,
                        MessageCode := 0,
                        MessageText := 'Command.Reserve3 = {1}',
                        Para1       :=  BYTE_TO_STRING(_command.Reserve3));

// Create log entry for MoveTime
CreateLogMessagePara1 ( Timestamp   := AxesGroup.InternalData.SystemTime,
                        MessageType := MessageType.CMD,
                        Severity    := Severity.DEBUG,
                        MessageCode := 0,
                        MessageText := 'Command.MoveTime = {1}',
                        Para1       :=  UINT_TO_STRING(_command.MoveTime));

// Create log entry for Position.E2
CreateLogMessagePara1 ( Timestamp   := AxesGroup.InternalData.SystemTime,
                        MessageType := MessageType.CMD,
                        Severity    := Severity.DEBUG,
                        MessageCode := 0,
                        MessageText := 'Command.Position.E2 = {1}',
                        Para1       :=  REAL_TO_STRING(_command.Position.E2));

// Create log entry for Position.E3
CreateLogMessagePara1 ( Timestamp   := AxesGroup.InternalData.SystemTime,
                        MessageType := MessageType.CMD,
                        Severity    := Severity.DEBUG,
                        MessageCode := 0,
                        MessageText := 'Command.Position.E3 = {1}',
                        Para1       :=  REAL_TO_STRING(_command.Position.E3));

// Create log entry for Position.E4
CreateLogMessagePara1 ( Timestamp   := AxesGroup.InternalData.SystemTime,
                        MessageType := MessageType.CMD,
                        Severity    := Severity.DEBUG,
                        MessageCode := 0,
                        MessageText := 'Command.Position.E4 = {1}',
                        Para1       :=  REAL_TO_STRING(_command.Position.E4));

// Create log entry for Position.E5
CreateLogMessagePara1 ( Timestamp   := AxesGroup.InternalData.SystemTime,
                        MessageType := MessageType.CMD,
                        Severity    := Severity.DEBUG,
                        MessageCode := 0,
                        MessageText := 'Command.Position.E5 = {1}',
                        Para1       :=  REAL_TO_STRING(_command.Position.E5));

// Create log entry for Position.E6
CreateLogMessagePara1 ( Timestamp   := AxesGroup.InternalData.SystemTime,
                        MessageType := MessageType.CMD,
                        Severity    := Severity.DEBUG,
                        MessageCode := 0,
                        MessageText := 'Command.Position.E6 = {1}',
                        Para1       :=  REAL_TO_STRING(_command.Position.E6));
END_METHOD

METHOD FB_init : BOOL
VAR_INPUT
  /// if TRUE, the retain variables are initialized (warm start / cold start)
  bInitRetains : BOOL; 
  /// if TRUE, the instance afterwards gets moved into the copy code (online change)
  bInCopyCode  : BOOL;  
END_VAR
MyType := 'MC_MoveLinearAbsoluteFB';
END_METHOD

METHOD PROTECTED OnCall
VAR_IN_OUT
  /// Robot assignment of function
  AxesGroup : AxesGroup; 
END_VAR
// call base implementation
SUPER^.OnCall(AxesGroup := AxesGroup);

CASE _stepCmd OF
  
  00:  IF ( _execute_R.Q )  
       THEN
         // Check function is supported and parameter are valid ?
         IF (( CheckFunctionSupported( AxesGroup := AxesGroup )) AND
             ( CheckParameterValid   ( AxesGroup := AxesGroup )))      
         THEN
           // set busy flag
           Busy := TRUE;
           // Reset command outputs
           SysDepMemSet(pDest := ADR(OutCmd), Value := 0, DataLen := SIZEOF(OutCmd));         
           // apply command parameter
          _parCmd := ParCmd;
           // init parameter sequence
          _command.ParSeq := 1;
           // create command data
           CommandData := CreateCommandPayload(AxesGroup := AxesGroup);
           // Add command to active command register
          _uniqueID := AxesGroup.Acyclic.ActiveCommandRegister.AddCmd( pCommandFB := ADR(THIS^ ));     
           // set timeout
           SetTimeout(PT := _timeoutCmd, rTimer := _timerCmd);
           // inc step counter
          _stepCmd := _stepCmd + 1;
         END_IF 
       END_IF
     

  01:  // Wait for responce received
       IF ( _responseReceived )
       THEN
         // reset response received flag
        _responseReceived := FALSE;
         // reset Active flag
         Active := FALSE;
         
         CASE  _response.State 
         OF
           CmdMessageState.BUFFERED    : CommandBuffered    := TRUE;
           CmdMessageState.ACTIVE      : Active             := TRUE;
           CmdMessageState.INTERRUPTED : CommandInterrupted := TRUE;           
           CmdMessageState.DONE        : Done               := TRUE;           
           CmdMessageState.ABORTED     : CommandAborted     := TRUE;
           CmdMessageState.ERROR       : Error              := TRUE;
         END_CASE
                
         // Done, Aborted or Error ?
         IF (_response.State >= CmdMessageState.DONE )
         THEN
           // Reset Busy flag
           Busy := FALSE;
           // Update results
           OutCmd.Progress          := _response.Progress;
           OutCmd.FollowID          := _response.OriginID;
           OutCmd.RemainingDistance := _response.RemainingDistance;
           // set timeout
           SetTimeout(PT := _timeoutCmd, rTimer := _timerCmd);
           // inc step counter
          _stepCmd := _stepCmd + 1; 
         END_IF
       END_IF


  02: IF ( NOT Execute)
      THEN
        Reset();
      END_IF     
      
ELSE
  // invalid step
  ErrorID := RobotLibraryEvents.ERR_INVALID_STEP;
END_CASE


// Reset FB
IF ( NOT Execute )
THEN
  Reset();
END_IF
END_METHOD

METHOD INTERNAL ParseResponsePayload : DINT
VAR_INPUT
  /// Response data
  ResponseData : RobotLibraryRecvDataFB;
  /// Timestamp
  Timestamp    : SystemTime;  
END_VAR
// Table 6-298: Received CMD payload (RC to PLC) of "MoveDirectRelative"
// --------------------------
// Header
// --------------------------
// Byte 00 : USINT   - ParSeq | State     
// Byte 01 : SINT    - AlarmMessageSeverity    
// Byte 02 : UINT    - AlarmMessageCode HB
// Byte 03 :         - AlarmMessageCode LB
// --------------------------
// Datablock
// --------------------------
// Byte 04 : USINT   - InvocationCounter
// Byte 05 : SINT    - Reserved
// Byte 06 : INT     - OriginID HW HB
// Byte 07 :         - OriginID HW LB
// Byte 08 : UINT    - Progress HW HB
// Byte 09 :         - Progress HW LB
// Byte 10 : REAL    - RemainingDistance HW HB
// Byte 11 :         - RemainingDistance HW LB
// Byte 12 :         - RemainingDistance LW HB
// Byte 13 :         - RemainingDistance LW LB
// call base implementation to parse the header from payload buffer
ResponseData.PayloadPtr := SUPER^.ParseResponsePayload(ResponseData := ResponseData, Timestamp := Timestamp);

// copy parsed header to response
_response.ParSeq               := _rspHeader.ParSeq;
_response.State                := _rspHeader.State;
_response.AlarmMessageSeverity := _rspHeader.AlarmMessageSeverity;
_response.AlarmMessageCode     := _rspHeader.AlarmMessageCode;

// Get Response.InvocationCounter
_response.InvocationCounter := ResponseData.GetUsint();
// Get Response.Reserve
_response.Reserve := ResponseData.GetSint();
// Get Response.OriginID
_response.OriginID := ResponseData.GetInt();
// Get Response.Progress
_response.Progress := ResponseData.GetUint();
// Get Response.RemainingDistance
_response.RemainingDistance := ResponseData.GetReal();

// Create logging
ParseResponsePayloadLog(ResponseData := ResponseData, Timestamp := Timestamp);
END_METHOD

METHOD INTERNAL ParseResponsePayloadLog
VAR_INPUT
  /// Response data
  ResponseData : RobotLibraryRecvDataFB;
  /// Timestamp
  Timestamp    : SystemTime;  
END_VAR
// Create log entry for Parameter start
CreateLogMessage      ( Timestamp   := Timestamp,
                        MessageType := MessageType.CMD,
                        Severity    := Severity.DEBUG,
                        MessageCode := 0,
                        MessageText := 'Parsed the following parameter(s) from response data:');
                        
// Create log entry for InvocationCounter
CreateLogMessagePara1 ( Timestamp   := Timestamp,
                        MessageType := MessageType.CMD,
                        Severity    := Severity.DEBUG,
                        MessageCode := 0,
                        MessageText := 'Response.InvocationCounter = {1}',
                        Para1       :=  USINT_TO_STRING(_response.InvocationCounter));

// Create log entry for Reserve
CreateLogMessagePara1 ( Timestamp   := Timestamp,
                        MessageType := MessageType.CMD,
                        Severity    := Severity.DEBUG,
                        MessageCode := 0,
                        MessageText := 'Response.Reserve = {1}',
                        Para1       :=  SINT_TO_STRING(_response.Reserve));

// Create log entry for OriginID
CreateLogMessagePara1 ( Timestamp   := Timestamp,
                        MessageType := MessageType.CMD,
                        Severity    := Severity.DEBUG,
                        MessageCode := 0,
                        MessageText := 'Response.OriginID = {1}',
                        Para1       :=  INT_TO_STRING(_response.OriginID));

// Create log entry for Progress
CreateLogMessagePara1 ( Timestamp   := Timestamp,
                        MessageType := MessageType.CMD,
                        Severity    := Severity.DEBUG,
                        MessageCode := 0,
                        MessageText := 'Response.Progress = {1}',
                        Para1       :=  UINT_TO_STRING(_response.Progress));

// Create log entry for RemainingDistance
CreateLogMessagePara1 ( Timestamp   := Timestamp,
                        MessageType := MessageType.CMD,
                        Severity    := Severity.DEBUG,
                        MessageCode := 0,
                        MessageText := 'Response.RemainingDistance = {1}',
                        Para1       :=  REAL_TO_STRING(_response.RemainingDistance));
END_METHOD

METHOD PROTECTED Reset : DINT
VAR_INPUT
END_VAR
Reset := SUPER^.Reset();

Done               := FALSE;
Busy               := FALSE;
Active             := FALSE;
CommandBuffered    := FALSE;
CommandAborted     := FALSE;
CommandInterrupted := FALSE;
END_METHOD

END_FUNCTION_BLOCK

// Library/POUs/BasicMove/MC_ReturnToPrimary/MC_ReturnToPrimaryFB
/// Return to path left during active interrupt
FUNCTION_BLOCK MC_ReturnToPrimaryFB EXTENDS RobotLibraryBaseFB
// ------------------------------------------------------------------------- 
//  SRCI Robot Library                                                
// ------------------------------------------------------------------------- 
//                                                                           
//  Object:      ReturnToPrimaryFB                                       
//  Author:      Thorsten Brach                                                
//  Date:        2024-06-01
//
//  Description:                                              
//   
//                                                                           
//  Copyright: 
//    (C) 2024 Thorsten Brach. All rights reserved                                                                                                                                            
//             Licensed under the LGPL-3.0 license.
//                                                                           
//  Disclaimer:                                                                           
//    This project is provided without any guarantee and can be used for   
//    private and commercial purposes. Any use is at the user’s 
//    own risk and responsibility.
//
// -------------------------------------------------------------------------
VAR_INPUT
  /// Activate ReturnToPrimary
  Enable             : BOOL;
  /// command parameter
  ParCmd             : ReturnToPrimaryParCmd;      
END_VAR

VAR_OUTPUT
  /// The command has been completed successfully
  Done               : BOOL;
  /// FB is being processed
  Busy               : BOOL;
  /// Command is transferred and confirmed by the RC
  CommandBuffered    : BOOL;
  /// The command takes control of the motion of the according axis group
  Active             : BOOL;
  /// The command was aborted by another command.
  CommandAborted     : BOOL;
  /// TRUE, while command is interrupted during execution and can be continued
  CommandInterrupted : BOOL;
  /// command results
  OutCmd             : ReturnToPrimaryOutCmd;      
END_VAR

VAR
  /// internal copy of command parameter 
 _parCmd             : ReturnToPrimaryParCmd;
  /// command data to send
 _command            : ReturnToPrimarySendData;
  /// response data received
 _response           : ReturnToPrimaryRecvData;      
  /// Rising edge for enable
 _enable_R           : R_TRIG;
  /// Falling edge for enable
 _enable_F           : F_TRIG;
END_VAR

SUPER^(AxesGroup := AxesGroup);

METHOD PROTECTED CheckFunctionSupported : BOOL
VAR_IN_OUT
  /// Robot assignment of function
  AxesGroup : AxesGroup; 
END_VAR
CheckFunctionSupported := AxesGroup.InternalData.RCSupportedFunctions.ReturnToPrimary;

IF ( NOT CheckFunctionSupported )
THEN
  // call base implementation for set error and create log entry
  SUPER^.CheckFunctionSupported(AxesGroup := AxesGroup);
END_IF
END_METHOD

METHOD PROTECTED CheckParameterChanged : BOOL
VAR_IN_OUT
  /// Robot assignment of function
  AxesGroup    : AxesGroup; 
END_VAR
// Check ParCmd Size is > 0, because MemCmp does not work correctly with size = 0
IF (SIZEOF(ParCmd) = 0) 
THEN 
  RETURN;
END_IF

// compare memory 
_parameterChanged := ( SysDepMemCmp(pData1 := ADR(ParCmd), pData2 := ADR(_parCmd), DataLen := SIZEOF(ParCmd)) <> RobotLibraryConstants.OK );

// check parameter valid ?
_parameterValid   := CheckParameterValid( AxesGroup := AxesGroup );

IF ((  _parameterChanged        )  AND 
    (  _parameterValid          )) OR
    (  _parameterUpdateInternal )  
THEN  
  // reset internal flag for send parameter update
 _parameterUpdateInternal := FALSE;
  // update internal copy of parameters 
 _parCmd := ParCmd;
  // inc parameter sequence
 _command.ParSeq := _command.ParSeq + 1;
  // update command data  
  CommandData := CreateCommandPayload(AxesGroup := AxesGroup); // ( Access via reference to rCommandFB in ACR )
  // notify active command register 
  AxesGroup.Acyclic.ActiveCommandRegister.NotifyParameterChanged := _uniqueID;
END_IF
END_METHOD

METHOD INTERNAL CreateCommandPayload : RobotLibrarySendDataFB
VAR_IN_OUT
  /// Robot assignment of function
  AxesGroup : AxesGroup; 
END_VAR
// Table 6-310: Sent CMD payload (PLC to RC) of "ReturnToPrimary"
// --------------------------
// Header
// --------------------------
// Byte 00 : UINT  - Type HB     
// Byte 01 :       - Type LB    
// Byte 02 : USINT - Reserve | ExecutionMode
// Byte 03 : USINT - ParSeq  | Priority
// --------------------------
// Datablock
// --------------------------
// Byte 04  : UINT  - ToolNo LW HB
// Byte 05  :       - ToolNo LW LB
// Byte 06  : UINT  - FrameNo LW HB
// Byte 07  :       - FrameNo LW LB
// Byte 08  : UINT  - VelocityRate LW HB
// Byte 09  :       - VelocityRate LW LB
// Byte 10  : UINT  - AccelerationRate LW HB
// Byte 11  :       - AccelerationRate LW LB
// Byte 12  : UINT  - DecelerationRate LW HB
// Byte 13  :       - DecelerationRate LW LB
// Byte 14  : UINT  - JerkRate LW HB
// Byte 15  :       - JerkRate LW LB
// Byte 16  : REAL  - Limit HW HB
// Byte 17  :       - Limit HW LB
// Byte 18  :       - Limit LW HB
// Byte 19  :       - Limit LW LB
// Byte 20  : BOOL  - ReturnMode
// Byte 21  : BOOL  - TrajectoryMode
// Byte 22  : UINT  - Time LW HB
// Byte 23  : UINT  - Time LW LB


// --------------------------
// set command parameter 
_command.CmdTyp            :=  CmdType.ReturnToPrimary;
_command.ExecMode          :=  ExecMode;
_command.ParSeq            := _command.ParSeq;
_command.Priority          :=  Priority;
_command.ToolNo            := _parCmd.ToolNo;
_command.FrameNo           := _parCmd.FrameNo;
_command.VelocityRate      :=  REAL_TO_PERCENT_UINT(_parCmd.VelocityRate     , IsOptional := FALSE);
_command.AccelerationRate  :=  REAL_TO_PERCENT_UINT(_parCmd.AccelerationRate , IsOptional := FALSE);
_command.DecelerationRate  :=  REAL_TO_PERCENT_UINT(_parCmd.DecelerationRate , IsOptional := TRUE );
_command.JerkRate          :=  REAL_TO_PERCENT_UINT(_parCmd.JerkRate         , IsOptional := TRUE );
_command.DistanceLimit     := _parCmd.DistanceLimit;
_command.ReturnMode        :=(_parCmd.ReturnMode = ReturnMode.END_POSITION);
_command.TrajectoryMode    := _parCmd.TrajectoryMode = TrajectoryMode.PTP_MOVEMENT;
_command.MoveTime          :=  TIME_TO_UINT(_parCmd.MoveTime);


// copy command data to header
_cmdHeader := _command;
// call base implementation to copy header to payload buffer
CreateCommandPayload := SUPER^.CreateCommandPayload(AxesGroup := AxesGroup);

// add command.ToolNo
CreateCommandPayload.AddUint(_command.ToolNo);
// add command.FrameNo
CreateCommandPayload.AddUint(_command.FrameNo);
// add command.VelocityRate
CreateCommandPayload.AddUint(_command.VelocityRate);
// add command.AccelerationRate
CreateCommandPayload.AddUint(_command.AccelerationRate);
// add command.DecelerationRate
CreateCommandPayload.AddUint(_command.DecelerationRate);
// add command.JerkRate
CreateCommandPayload.AddUint(_command.JerkRate);
// add command.DistanceLimit
CreateCommandPayload.AddReal(_command.DistanceLimit);
// add command.ReturnMode
CreateCommandPayload.AddBool(_command.ReturnMode);
// add command.TrajectoryMode
CreateCommandPayload.AddBool(_command.TrajectoryMode);
// add command.MoveTime
CreateCommandPayload.AddUint(_command.MoveTime);

// Create logging
CreateCommandPayloadLog(AxesGroup := AxesGroup);
END_METHOD

METHOD INTERNAL CreateCommandPayloadLog 
VAR_IN_OUT
  /// Robot assignment of function
  AxesGroup : AxesGroup; 
END_VAR
// Create log entry for Parameter start
CreateLogMessage      ( Timestamp   := AxesGroup.InternalData.SystemTime,
                        MessageType := MessageType.CMD,
                        Severity    := Severity.DEBUG,
                        MessageCode := 0,
                        MessageText := 'Create command payload with the following parameter(s) :');

// Create log entry for ToolNo
CreateLogMessagePara1 ( Timestamp   := AxesGroup.InternalData.SystemTime,
                        MessageType := MessageType.CMD,
                        Severity    := Severity.DEBUG,
                        MessageCode := 0,
                        MessageText := 'Command.ToolNo = {1}',
                        Para1       :=  USINT_TO_STRING(_command.ToolNo));

// Create log entry for FrameNo
CreateLogMessagePara1 ( Timestamp   := AxesGroup.InternalData.SystemTime,
                        MessageType := MessageType.CMD,
                        Severity    := Severity.DEBUG,
                        MessageCode := 0,
                        MessageText := 'Command.FrameNo = {1}',
                        Para1       :=  USINT_TO_STRING(_command.FrameNo));

// Create log entry for VelocityRate
CreateLogMessagePara1 ( Timestamp   := AxesGroup.InternalData.SystemTime,
                        MessageType := MessageType.CMD,
                        Severity    := Severity.DEBUG,
                        MessageCode := 0,
                        MessageText := 'Command.VelocityRate = {1}',
                        Para1       :=  UINT_TO_STRING(_command.VelocityRate));

// Create log entry for AccelerationRate
CreateLogMessagePara1 ( Timestamp   := AxesGroup.InternalData.SystemTime,
                        MessageType := MessageType.CMD,
                        Severity    := Severity.DEBUG,
                        MessageCode := 0,
                        MessageText := 'Command.AccelerationRate = {1}',
                        Para1       :=  UINT_TO_STRING(_command.AccelerationRate));
                        
// Create log entry for DecelerationRate
CreateLogMessagePara1 ( Timestamp   := AxesGroup.InternalData.SystemTime,
                        MessageType := MessageType.CMD,
                        Severity    := Severity.DEBUG,
                        MessageCode := 0,
                        MessageText := 'Command.DecelerationRate = {1}',
                        Para1       :=  UINT_TO_STRING(_command.DecelerationRate));

// Create log entry for JerkRate
CreateLogMessagePara1 ( Timestamp   := AxesGroup.InternalData.SystemTime,
                        MessageType := MessageType.CMD,
                        Severity    := Severity.DEBUG,
                        MessageCode := 0,
                        MessageText := 'Command.JerkRate = {1}',
                        Para1       :=  UINT_TO_STRING(_command.JerkRate));

// Create log entry for DistanceLimit
CreateLogMessagePara1 ( Timestamp   := AxesGroup.InternalData.SystemTime,
                        MessageType := MessageType.CMD,
                        Severity    := Severity.DEBUG,
                        MessageCode := 0,
                        MessageText := 'Command.DistanceLimit = {1}',
                        Para1       :=  REAL_TO_STRING(_command.DistanceLimit));

// Create log entry for ReturnMode
CreateLogMessagePara1 ( Timestamp   := AxesGroup.InternalData.SystemTime,
                        MessageType := MessageType.CMD,
                        Severity    := Severity.DEBUG,
                        MessageCode := 0,
                        MessageText := 'Command.ReturnMode = {1}',
                        Para1       :=  BOOL_TO_STRING(_command.ReturnMode));

// Create log entry for TrajectoryMode
CreateLogMessagePara1 ( Timestamp   := AxesGroup.InternalData.SystemTime,
                        MessageType := MessageType.CMD,
                        Severity    := Severity.DEBUG,
                        MessageCode := 0,
                        MessageText := 'Command.TrajectoryMode = {1}',
                        Para1       :=  BOOL_TO_STRING(_command.TrajectoryMode));

// Create log entry for MoveTime
CreateLogMessagePara1 ( Timestamp   := AxesGroup.InternalData.SystemTime,
                        MessageType := MessageType.CMD,
                        Severity    := Severity.DEBUG,
                        MessageCode := 0,
                        MessageText := 'Command.MoveTime = {1}',
                        Para1       :=  UINT_TO_STRING(_command.MoveTime));
END_METHOD

METHOD FB_init : BOOL
VAR_INPUT
  /// if TRUE, the retain variables are initialized (warm start / cold start)
  bInitRetains : BOOL; 
  /// if TRUE, the instance afterwards gets moved into the copy code (online change)
  bInCopyCode  : BOOL;  
END_VAR
MyType := 'MC_ReturnToPrimaryFB';
END_METHOD

METHOD PROTECTED OnCall
VAR_IN_OUT
  /// Robot assignment of function
  AxesGroup : AxesGroup; 
END_VAR
// call base implementation
SUPER^.OnCall(AxesGroup := AxesGroup);

// building rising and falling edges
_enable_R( CLK := Enable);
_enable_F( CLK := Enable);

CASE _stepCmd OF
  
  00:  IF ( _enable_R.Q )  
       THEN
         // reset the rising edge
        _enable_R();       
         // reset the falling edge
        _enable_F();   
    
         // Check function is supported and parameter are valid ?
         IF (( CheckFunctionSupported( AxesGroup := AxesGroup )) AND
             ( CheckParameterValid   ( AxesGroup := AxesGroup )))      
         THEN
           // set busy flag
           Busy := TRUE;
           // Reset command outputs
           SysDepMemSet(pDest := ADR(OutCmd), Value := 0, DataLen := SIZEOF(OutCmd));         
           // apply command parameter
          _parCmd := ParCmd;
           // init parameter sequence
          _command.ParSeq := 1;
           // create command data
           CommandData := CreateCommandPayload(AxesGroup := AxesGroup);
           // Add command to active command register
          _uniqueID := AxesGroup.Acyclic.ActiveCommandRegister.AddCmd( pCommandFB := ADR(THIS^ ));     
           // set timeout
           SetTimeout(PT := _timeoutCmd, rTimer := _timerCmd);
           // inc step counter
          _stepCmd := _stepCmd + 1;
         END_IF 
       END_IF
     

  01:  // Wait for responce received
       IF ( _responseReceived )
       THEN
         // reset response received flag
        _responseReceived := FALSE;
         // reset Active flag
         Active := FALSE;
         
         CASE  _response.State 
         OF
           CmdMessageState.BUFFERED    : CommandBuffered    := TRUE;
           CmdMessageState.ACTIVE      : Active             := TRUE;
           CmdMessageState.INTERRUPTED : CommandInterrupted := TRUE;
           CmdMessageState.DONE        : Done               := TRUE;
           CmdMessageState.ABORTED     : CommandAborted     := TRUE;
           CmdMessageState.ERROR       : Error              := TRUE;
         END_CASE
                
         // Done, Aborted or Error ?
         IF (_response.State >= CmdMessageState.DONE )
         THEN
           // Reset Busy flag
           Busy := FALSE;
           // Update results
           OutCmd.Progress          := _response.Progress;
           OutCmd.RemainingDistance := _response.RemainingDistance;
           OutCmd.PrimaryPosToolNo  := UINT_TO_USINT(_response.PrimaryPosToolNo);  {warning 'ToDo'}
           OutCmd.PrimaryPosFrameNo := UINT_TO_USINT(_response.PrimaryPosFrameNo); {warning 'ToDo'}
           
           // set timeout
           SetTimeout(PT := _timeoutCmd, rTimer := _timerCmd);
           // inc step counter
          _stepCmd := _stepCmd + 1; 
         END_IF
       END_IF


  02: IF (NOT Enable)
      THEN
        Reset();
      END_IF  

ELSE
  // invalid step
  ErrorID := RobotLibraryEvents.ERR_INVALID_STEP;
END_CASE



// Reset FB
IF (( _enable_R.Q ) OR
    ( _enable_F.Q ))
THEN
  Reset();
END_IF
END_METHOD

METHOD INTERNAL ParseResponsePayload : DINT
VAR_INPUT
  /// Response data
  ResponseData : RobotLibraryRecvDataFB;
  /// Timestamp
  Timestamp    : SystemTime;  
END_VAR
// Table 6-311: Received CMD payload (RC to PLC) of "ReturnToPrimary"
// --------------------------
// Header
// --------------------------
// Byte 00 : USINT - ParSeq | State     
// Byte 01 : SINT  - AlarmMessageSeverity    
// Byte 02 : UINT  - AlarmMessageCode HB
// Byte 03 :       - AlarmMessageCode LB
// --------------------------
// Datablock
// --------------------------
// Byte 04 : UINT  - Progress LW HB
// Byte 05 :       - Progress LW LB
// Byte 06 : REAL  - RemainingDistance HW HB
// Byte 07 :       - RemainingDistance HW LB
// Byte 08 :       - RemainingDistance LW HB
// Byte 09 :       - RemainingDistance LW LB
// Byte 10 : UINT  - PrimaryPosToolNo LW HB
// Byte 11 :       - PrimaryPosToolNo LW LB
// --------------------------
// call base implementation to parse the header from payload buffer
ResponseData.PayloadPtr := SUPER^.ParseResponsePayload(ResponseData := ResponseData, Timestamp := Timestamp);

// copy parsed header to response
_response.ParSeq               := _rspHeader.ParSeq;
_response.State                := _rspHeader.State;
_response.AlarmMessageSeverity := _rspHeader.AlarmMessageSeverity;
_response.AlarmMessageCode     := _rspHeader.AlarmMessageCode;

// Get Response.Progress
_response.Progress             := ResponseData.GetUint();
// Get Response.RemainingDistance
_response.RemainingDistance    := ResponseData.GetReal();
// Get Response.PrimaryPosToolNo
_response.PrimaryPosToolNo     := ResponseData.GetUint();
// Get Response.PrimaryPosFrameNo
_response.PrimaryPosFrameNo    := ResponseData.GetUint();

// Create logging
ParseResponsePayloadLog(ResponseData := ResponseData, Timestamp := Timestamp);
END_METHOD

METHOD INTERNAL ParseResponsePayloadLog
VAR_INPUT
  /// Response data
  ResponseData : RobotLibraryRecvDataFB;
  /// Timestamp
  Timestamp    : SystemTime;  
END_VAR
// Create log entry for Parameter start
CreateLogMessage      ( Timestamp   := Timestamp,
                        MessageType := MessageType.CMD,
                        Severity    := Severity.DEBUG,
                        MessageCode := 0,
                        MessageText := 'Parsed the following parameter(s) from response data:');
                        
// Create log entry for Progress
CreateLogMessagePara1 ( Timestamp   := Timestamp,
                        MessageType := MessageType.CMD,
                        Severity    := Severity.DEBUG,
                        MessageCode := 0,
                        MessageText := 'Response.Progress = {1}',
                        Para1       :=  UINT_TO_STRING(_response.Progress));

// Create log entry for RemainingDistance
CreateLogMessagePara1 ( Timestamp   := Timestamp,
                        MessageType := MessageType.CMD,
                        Severity    := Severity.DEBUG,
                        MessageCode := 0,
                        MessageText := 'Response.RemainingDistance = {1}',
                        Para1       :=  REAL_TO_STRING(_response.RemainingDistance));

// Create log entry for PrimaryPosToolNo
CreateLogMessagePara1 ( Timestamp   := Timestamp,
                        MessageType := MessageType.CMD,
                        Severity    := Severity.DEBUG,
                        MessageCode := 0,
                        MessageText := 'Response.PrimaryPosToolNo = {1}',
                        Para1       :=  UINT_TO_STRING(_response.PrimaryPosToolNo));

// Create log entry for PrimaryPosFrameNo
CreateLogMessagePara1 ( Timestamp   := Timestamp,
                        MessageType := MessageType.CMD,
                        Severity    := Severity.DEBUG,
                        MessageCode := 0,
                        MessageText := 'Response.PrimaryPosFrameNo = {1}',
                        Para1       :=  UINT_TO_STRING(_response.PrimaryPosFrameNo));
END_METHOD

METHOD PROTECTED Reset : DINT
VAR_INPUT
END_VAR
Reset := SUPER^.Reset();

Done               := FALSE;
Busy               := FALSE;
Active             := FALSE;
CommandBuffered    := FALSE;
CommandAborted     := FALSE;
CommandInterrupted := FALSE;
END_METHOD

END_FUNCTION_BLOCK

// Library/POUs/Calculation/MC_CalculateCartesianPosition/MC_CalculateCartesianPositionFB
/// Calculate cartesian position from existing cartesian position
FUNCTION_BLOCK MC_CalculateCartesianPositionFB EXTENDS RobotLibraryBaseExecuteFB
// ------------------------------------------------------------------------- 
//  SRCI Robot Library                                                
// ------------------------------------------------------------------------- 
//                                                                           
//  Object:      CalculateCartesianPositionFB                                       
//  Author:      Thorsten Brach                                                
//  Date:        2024-06-01
//
//  Description:                                              
//   
//                                                                           
//  Copyright: 
//    (C) 2024 Thorsten Brach. All rights reserved                                                                                                                                            
//             Licensed under the LGPL-3.0 license.
//                                                                           
//  Disclaimer:                                                                           
//    This project is provided without any guarantee and can be used for   
//    private and commercial purposes. Any use is at the user’s 
//    own risk and responsibility.
//
// -------------------------------------------------------------------------
VAR_INPUT
  /// Command parameter 
  ParCmd          : CalculateCartesianPositionParCmd;  
END_VAR

VAR_OUTPUT
  /// Command is transferred and confirmed by the RC
  CommandBuffered : BOOL;
  /// Command output 
  OutCmd          : CalculateCartesianPositionOutCmd;  
END_VAR

VAR
  /// internal copy of command parameter 
 _parCmd          : CalculateCartesianPositionParCmd;
  /// command data to send
 _command         : CalculateCartesianPositionSendData;
  /// response data received
 _response        : CalculateCartesianPositionRecvData;      
END_VAR

SUPER^(AxesGroup := AxesGroup);

METHOD PROTECTED CheckFunctionSupported : BOOL
VAR_IN_OUT
  /// Robot assignment of function
  AxesGroup : AxesGroup; 
END_VAR
CheckFunctionSupported := AxesGroup.InternalData.RCSupportedFunctions.CalculateCartesianPosition;

IF ( NOT CheckFunctionSupported )
THEN
  // call base implementation for set error and create log entry
  SUPER^.CheckFunctionSupported(AxesGroup := AxesGroup);
END_IF
END_METHOD

METHOD PROTECTED CheckParameterChanged : BOOL
VAR_IN_OUT
  /// Robot assignment of function
  AxesGroup    : AxesGroup; 
END_VAR
// Check ParCmd Size is > 0, because MemCmp does not work correctly with size = 0
IF (SIZEOF(ParCmd) = 0) 
THEN 
  RETURN;
END_IF

// compare memory 
_parameterChanged := ( SysDepMemCmp(pData1 := ADR(ParCmd), pData2 := ADR(_parCmd), DataLen := SIZEOF(ParCmd)) <> RobotLibraryConstants.OK );

// check parameter valid ?
_parameterValid   := CheckParameterValid( AxesGroup := AxesGroup );

IF ((  _parameterChanged        )  AND 
    (  _parameterValid          )) OR
    (  _parameterUpdateInternal )  
THEN  
  // reset internal flag for send parameter update
 _parameterUpdateInternal := FALSE;
  // update internal copy of parameters 
 _parCmd := ParCmd;
  // inc parameter sequence
 _command.ParSeq := _command.ParSeq + 1;
  // update command data  
  CommandData := CreateCommandPayload(AxesGroup := AxesGroup); // ( Access via reference to rCommandFB in ACR )
  // notify active command register 
  AxesGroup.Acyclic.ActiveCommandRegister.NotifyParameterChanged := _uniqueID;
END_IF
END_METHOD

METHOD INTERNAL CreateCommandPayload : RobotLibrarySendDataFB
VAR_IN_OUT
  /// Robot assignment of function
  AxesGroup : AxesGroup; 
END_VAR
// Table 6-645: Received CMD payload (RC to PLC) of "CalculateCartesianPosition"
// --------------------------
// Header
// --------------------------
// Byte 00 : UINT       - Type HB     
// Byte 01 :            - Type LB    
// Byte 02 : USINT      - Reserve | ExecutionMode
// Byte 03 : USINT      - ParSeq  | Priority
// --------------------------
// Datablock
// --------------------------
// Byte 04 : USINT      - FrameNo
// Byte 05 : USINT      - TargetFrameNo
// Byte 06 : REAL       - Position.X  HW HB
// Byte 07 :            - Position.X  HW LB
// Byte 08 :            - Position.X  LW HB
// Byte 09 :            - Position.X  LW LB
// Byte 10 : REAL       - Position.Y  HW HB
// Byte 11 :            - Position.Y  HW LB
// Byte 12 :            - Position.Y  LW HB
// Byte 13 :            - Position.Y  LW LB
// Byte 14 : REAL       - Position.Z  HW HB
// Byte 15 :            - Position.Z  HW LB
// Byte 16 :            - Position.Z  LW HB
// Byte 17 :            - Position.Z  LW LB
// Byte 18 : REAL       - Position.Rx HW HB
// Byte 19 :            - Position.Rx HW LB
// Byte 20 :            - Position.Rx LW HB
// Byte 21 :            - Position.Rx LW LB
// Byte 22 : REAL       - Position.Ry HW HB
// Byte 23 :            - Position.Ry HW LB
// Byte 24 :            - Position.Ry LW HB
// Byte 25 :            - Position.Ry LW LB
// Byte 26 : REAL       - Position.Rz HW HB
// Byte 27 :            - Position.Rz HW LB
// Byte 28 :            - Position.Rz LW HB
// Byte 29 :            - Position.Rz LW LB
// Byte 30 : Config     - ArmConfig   LW HB
// Byte 31 :            - ArmConfig   LW LB
// Byte 32 : TurnNumber - J1 + J2     LW HB
// Byte 33 :            - J3 + J4     LW LB
// Byte 34 :            - J5 + J6     LW LB
// Byte 35 :            - E1          LW LB
// Byte 36 : REAL       - Position.E1 HW HB
// Byte 37 :            - Position.E1 HW LB
// Byte 38 :            - Position.E1 LW HB
// Byte 39 :            - Position.E1 LW LB
// Byte 40 : REAL       - Position.E2 HW HB
// Byte 41 :            - Position.E2 HW LB
// Byte 42 :            - Position.E2 LW HB
// Byte 43 :            - Position.E2 LW LB
// Byte 44 : REAL       - Position.E3 HW HB
// Byte 45 :            - Position.E3 HW LB
// Byte 46 :            - Position.E3 LW HB
// Byte 47 :            - Position.E3 LW LB
// Byte 48 : REAL       - Position.E4 HW HB
// Byte 49 :            - Position.E4 HW LB
// Byte 50 :            - Position.E4 LW HB
// Byte 51 :            - Position.E4 LW LB
// Byte 52 : REAL       - Position.E5 HW HB
// Byte 53 :            - Position.E5 HW LB
// Byte 54 :            - Position.E5 LW HB
// Byte 55 :            - Position.E5 LW LB
// Byte 56 : REAL       - Position.E6 HW HB
// Byte 57 :            - Position.E6 HW LB
// Byte 58 :            - Position.E6 LW HB
// Byte 59 :            - Position.E6 LW LB
// --------------------------
// set command parameter 
_command.CmdTyp            :=  CmdType.CalculateCartesianPosition;
_command.ExecMode          :=  ExecMode;
_command.ParSeq            := _command.ParSeq;
_command.Priority          :=  Priority;
_command.FrameNo           := _parCmd.FrameNo;
_command.TargetFrameNo     := _parCmd.TargetFrameNo;
_command.CartesianPosition := _parCmd.CartesianPosition;

// copy command data to header
_cmdHeader := _command;
// call base implementation to copy header to payload buffer
CreateCommandPayload := SUPER^.CreateCommandPayload(AxesGroup := AxesGroup);

// add command.FrameNo
CreateCommandPayload.AddUsint(_command.FrameNo);
// add command.TargetFrameNo
CreateCommandPayload.AddUsint(_command.TargetFrameNo);
// add command.CartesianPosition.X
CreateCommandPayload.AddReal(_command.CartesianPosition.X);
// add command.CartesianPosition.Y
CreateCommandPayload.AddReal(_command.CartesianPosition.Y);
// add command.CartesianPosition.Z
CreateCommandPayload.AddReal(_command.CartesianPosition.Z);
// add command.CartesianPosition.Rx
CreateCommandPayload.AddReal(_command.CartesianPosition.Rx);
// add command.CartesianPosition.Ry
CreateCommandPayload.AddReal(_command.CartesianPosition.Ry);
// add command.CartesianPosition.Rz
CreateCommandPayload.AddReal(_command.CartesianPosition.Rz);
// add command.CartesianPosition.Config
CreateCommandPayload.AddArmConfig(_command.CartesianPosition.Config);
// add command.CartesianPosition.TurnNumber
CreateCommandPayload.AddTurnNumber(_command.CartesianPosition.TurnNumber);
// add command.CartesianPosition.E1
CreateCommandPayload.AddReal(_command.CartesianPosition.E1);
// add command.CartesianPosition.E2
CreateCommandPayload.AddReal(_command.CartesianPosition.E2);
// add command.CartesianPosition.E3
CreateCommandPayload.AddReal(_command.CartesianPosition.E3);
// add command.CartesianPosition.E4
CreateCommandPayload.AddReal(_command.CartesianPosition.E4);
// add command.CartesianPosition.E5
CreateCommandPayload.AddReal(_command.CartesianPosition.E5);
// add command.CartesianPosition.E6
CreateCommandPayload.AddReal(_command.CartesianPosition.E6);

// Create logging
CreateCommandPayloadLog(AxesGroup := AxesGroup);
END_METHOD

METHOD INTERNAL CreateCommandPayloadLog 
VAR_IN_OUT
  /// Robot assignment of function
  AxesGroup : AxesGroup; 
END_VAR
// Create log entry for Parameter start
CreateLogMessage      ( Timestamp   := AxesGroup.InternalData.SystemTime,
                        MessageType := MessageType.CMD,
                        Severity    := Severity.DEBUG,
                        MessageCode := 0,
                        MessageText := 'Create command payload with the following parameter(s) :');

// Create log entry for FrameNo
CreateLogMessagePara1 ( Timestamp   := AxesGroup.InternalData.SystemTime,
                        MessageType := MessageType.CMD,
                        Severity    := Severity.DEBUG,
                        MessageCode := 0,
                        MessageText := 'Command.FrameNo = {1}',
                        Para1       :=  USINT_TO_STRING(_command.FrameNo));

// Create log entry for TargetFrameNo
CreateLogMessagePara1 ( Timestamp   := AxesGroup.InternalData.SystemTime,
                        MessageType := MessageType.CMD,
                        Severity    := Severity.DEBUG,
                        MessageCode := 0,
                        MessageText := 'Command.TargetFrameNo = {1}',
                        Para1       :=  USINT_TO_STRING(_command.TargetFrameNo));

// Create log entry for CartesianPosition.X
CreateLogMessagePara1 ( Timestamp   := AxesGroup.InternalData.SystemTime,
                        MessageType := MessageType.CMD,
                        Severity    := Severity.DEBUG,
                        MessageCode := 0,
                        MessageText := 'Command.CartesianPosition.X = {1}',
                        Para1       :=  REAL_TO_STRING(_command.CartesianPosition.X));

// Create log entry for CartesianPosition.Y
CreateLogMessagePara1 ( Timestamp   := AxesGroup.InternalData.SystemTime,
                        MessageType := MessageType.CMD,
                        Severity    := Severity.DEBUG,
                        MessageCode := 0,
                        MessageText := 'Command.CartesianPosition.Y = {1}',
                        Para1       :=  REAL_TO_STRING(_command.CartesianPosition.Y));

// Create log entry for CartesianPosition.Z
CreateLogMessagePara1 ( Timestamp   := AxesGroup.InternalData.SystemTime,
                        MessageType := MessageType.CMD,
                        Severity    := Severity.DEBUG,
                        MessageCode := 0,
                        MessageText := 'Command.CartesianPosition.Z = {1}',
                        Para1       :=  REAL_TO_STRING(_command.CartesianPosition.Z));

// Create log entry for CartesianPosition.Rx
CreateLogMessagePara1 ( Timestamp   := AxesGroup.InternalData.SystemTime,
                        MessageType := MessageType.CMD,
                        Severity    := Severity.DEBUG,
                        MessageCode := 0,
                        MessageText := 'Command.CartesianPosition.Rx = {1}',
                        Para1       :=  REAL_TO_STRING(_command.CartesianPosition.Rx));

// Create log entry for CartesianPosition.Ry
CreateLogMessagePara1 ( Timestamp   := AxesGroup.InternalData.SystemTime,
                        MessageType := MessageType.CMD,
                        Severity    := Severity.DEBUG,
                        MessageCode := 0,
                        MessageText := 'Command.CartesianPosition.Ry = {1}',
                        Para1       :=  REAL_TO_STRING(_command.CartesianPosition.Ry));

// Create log entry for CartesianPosition.Rz
CreateLogMessagePara1 ( Timestamp   := AxesGroup.InternalData.SystemTime,
                        MessageType := MessageType.CMD,
                        Severity    := Severity.DEBUG,
                        MessageCode := 0,
                        MessageText := 'Command.CartesianPosition.Rz = {1}',
                        Para1       :=  REAL_TO_STRING(_command.CartesianPosition.Rz));

// Create log entry for CartesianPosition.Config
CreateLogMessagePara1 ( Timestamp   := AxesGroup.InternalData.SystemTime,
                        MessageType := MessageType.CMD,
                        Severity    := Severity.DEBUG,
                        MessageCode := 0,
                        MessageText := 'Command.CartesianPosition.Config = {1}',
                        Para1       :=  ARM_CONFIG_TO_STRING(_command.CartesianPosition.Config));

// Create log entry for CartesianPosition.TurnNumber[0]
CreateLogMessagePara1 ( Timestamp   := AxesGroup.InternalData.SystemTime,
                        MessageType := MessageType.CMD,
                        Severity    := Severity.DEBUG,
                        MessageCode := 0,
                        MessageText := 'Command.CartesianPosition.TurnNumber[0] = {1}',
                        Para1       :=  BYTE_TO_STRING(CombineHalfSints(HalfSintHi := _command.CartesianPosition.TurnNumber.J2Turns, 
                                                                        HalfSintLo := _command.CartesianPosition.TurnNumber.J1Turns)));

// Create log entry for CartesianPosition.TurnNumber[1]
CreateLogMessagePara1 ( Timestamp   := AxesGroup.InternalData.SystemTime,
                        MessageType := MessageType.CMD,
                        Severity    := Severity.DEBUG,
                        MessageCode := 0,
                        MessageText := 'Command.CartesianPosition.TurnNumber[1] = {1}',
                        Para1       :=  BYTE_TO_STRING(CombineHalfSints(HalfSintHi := _command.CartesianPosition.TurnNumber.J4Turns, 
                                                                        HalfSintLo := _command.CartesianPosition.TurnNumber.J3Turns)));

// Create log entry for CartesianPosition.TurnNumber[2]
CreateLogMessagePara1 ( Timestamp   := AxesGroup.InternalData.SystemTime,
                        MessageType := MessageType.CMD,
                        Severity    := Severity.DEBUG,
                        MessageCode := 0,
                        MessageText := 'Command.CartesianPosition.TurnNumber[2] = {1}',
                        Para1       :=  BYTE_TO_STRING(CombineHalfSints(HalfSintHi := _command.CartesianPosition.TurnNumber.J6Turns, 
                                                                        HalfSintLo := _command.CartesianPosition.TurnNumber.J5Turns)));

// Create log entry for CartesianPosition.TurnNumber[3]
CreateLogMessagePara1 ( Timestamp   := AxesGroup.InternalData.SystemTime,
                        MessageType := MessageType.CMD,
                        Severity    := Severity.DEBUG,
                        MessageCode := 0,
                        MessageText := 'Command.CartesianPosition.TurnNumber[3] = {1}',
                        Para1       :=  SINT_TO_STRING(_command.CartesianPosition.TurnNumber.E1Turns));

// Create log entry for CartesianPosition.E1
CreateLogMessagePara1 ( Timestamp   := AxesGroup.InternalData.SystemTime,
                        MessageType := MessageType.CMD,
                        Severity    := Severity.DEBUG,
                        MessageCode := 0,
                        MessageText := 'Command.CartesianPosition.E1 = {1}',
                        Para1       :=  REAL_TO_STRING(_command.CartesianPosition.E1));

// Create log entry for CartesianPosition.E2
CreateLogMessagePara1 ( Timestamp   := AxesGroup.InternalData.SystemTime,
                        MessageType := MessageType.CMD,
                        Severity    := Severity.DEBUG,
                        MessageCode := 0,
                        MessageText := 'Command.CartesianPosition.E2 = {1}',
                        Para1       :=  REAL_TO_STRING(_command.CartesianPosition.E2));

// Create log entry for CartesianPosition.E3
CreateLogMessagePara1 ( Timestamp   := AxesGroup.InternalData.SystemTime,
                        MessageType := MessageType.CMD,
                        Severity    := Severity.DEBUG,
                        MessageCode := 0,
                        MessageText := 'Command.CartesianPosition.E3 = {1}',
                        Para1       :=  REAL_TO_STRING(_command.CartesianPosition.E3));

// Create log entry for CartesianPosition.E4
CreateLogMessagePara1 ( Timestamp   := AxesGroup.InternalData.SystemTime,
                        MessageType := MessageType.CMD,
                        Severity    := Severity.DEBUG,
                        MessageCode := 0,
                        MessageText := 'Command.CartesianPosition.E4 = {1}',
                        Para1       :=  REAL_TO_STRING(_command.CartesianPosition.E4));

// Create log entry for CartesianPosition.E5
CreateLogMessagePara1 ( Timestamp   := AxesGroup.InternalData.SystemTime,
                        MessageType := MessageType.CMD,
                        Severity    := Severity.DEBUG,
                        MessageCode := 0,
                        MessageText := 'Command.CartesianPosition.E5 = {1}',
                        Para1       :=  REAL_TO_STRING(_command.CartesianPosition.E5));

// Create log entry for CartesianPosition.E6
CreateLogMessagePara1 ( Timestamp   := AxesGroup.InternalData.SystemTime,
                        MessageType := MessageType.CMD,
                        Severity    := Severity.DEBUG,
                        MessageCode := 0,
                        MessageText := 'Command.CartesianPosition.E6 = {1}',
                        Para1       :=  REAL_TO_STRING(_command.CartesianPosition.E6));
END_METHOD

METHOD FB_init : BOOL
VAR_INPUT
  /// if TRUE, the retain variables are initialized (warm start / cold start)
  bInitRetains : BOOL; 
  /// if TRUE, the instance afterwards gets moved into the copy code (online change)
  bInCopyCode  : BOOL;  
END_VAR
MyType := 'MC_CalculateCartesianPositionFB';

ExecMode := ExecutionMode.PARALLEL;
END_METHOD

METHOD PROTECTED OnCall
VAR_IN_OUT
  /// Robot assignment of function
  AxesGroup : AxesGroup; 
END_VAR
// call base implementation
SUPER^.OnCall(AxesGroup := AxesGroup);

CASE _stepCmd OF
  
  00:  IF ( _execute_R.Q )  
       THEN
         // Check function is supported and parameter are valid ?
         IF (( CheckFunctionSupported( AxesGroup := AxesGroup )) AND
             ( CheckParameterValid   ( AxesGroup := AxesGroup )))      
         THEN
           // set busy flag
           Busy := TRUE;
           // Reset command outputs
           SysDepMemSet(pDest := ADR(OutCmd), Value := 0, DataLen := SIZEOF(OutCmd));         
           // apply command parameter
          _parCmd := ParCmd;
           // init parameter sequence
          _command.ParSeq := 1;
           // create command data
           CommandData := CreateCommandPayload(AxesGroup := AxesGroup);
           // Add command to active command register
          _uniqueID := AxesGroup.Acyclic.ActiveCommandRegister.AddCmd( pCommandFB := ADR(THIS^ ));     
           // set timeout
           SetTimeout(PT := _timeoutCmd, rTimer := _timerCmd);
           // inc step counter
          _stepCmd := _stepCmd + 1; 
         END_IF
       END_IF
     

  01:  // Wait for responce received
       IF ( _responseReceived )
       THEN
         // reset response received flag
        _responseReceived := FALSE;

